// TIA Portal V20 export
TYPE "LER_typeCommonData"
// stored: Access Published
   STRUCT
      PartType : Byte;   // 1 = 100mm cell, 2 = 200mm cell, 3= gauge part , 4 = dry run
      PartStatus : Byte;   // 0: no part // 1: Parts available // 2 : Inspection busy // 3: OK // 4: NG
      LastMachineNumber : Byte;   // Last machine no: 20, 30, 60
      ProductionTimestamp : DTL;   // Time of last operation or machining
      Part_ID : String[32];   // Part ID
      ReworkRequested : Bool;   // Request to re-work
   END_STRUCT;
END_TYPE
